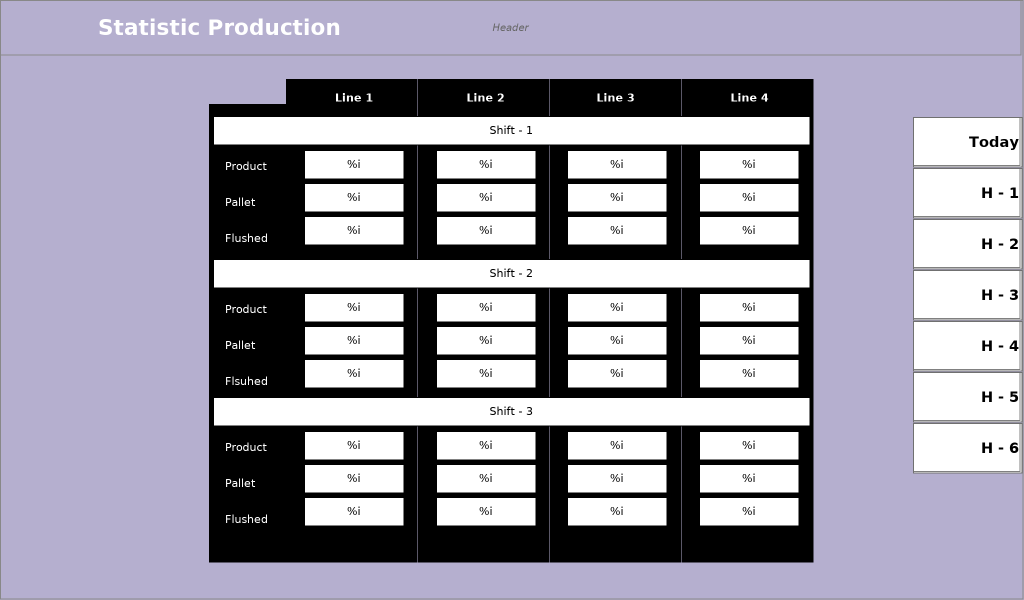
VISUALIZATION OEE_Counter  // 1024x600
    Frame (0,0 1021x55)
        shows Header()
    Button (913,117 109x50), "Today", image: VisuSymbols.Symbols.CalenderDay
        OnMouseClick: execute {
            Data_GVL.dt_OEECounter[1].HMI_NumberPrev := 0;
            Data_GVL.dt_OEECounter[2].HMI_NumberPrev := 0;
            Data_GVL.dt_OEECounter[3].HMI_NumberPrev := 0;
            Data_GVL.dt_OEECounter[4].HMI_NumberPrev := 0;
        }
    Button (913,168 109x50), "H - 1", image: VisuSymbols.Symbols.CalenderDay
        OnMouseClick: execute {
            Data_GVL.dt_OEECounter[1].HMI_NumberPrev := 1;
            Data_GVL.dt_OEECounter[2].HMI_NumberPrev := 1;
            Data_GVL.dt_OEECounter[3].HMI_NumberPrev := 1;
            Data_GVL.dt_OEECounter[4].HMI_NumberPrev := 1;
        }
    Button (913,219 109x50), "H - 2", image: VisuSymbols.Symbols.CalenderDay
        OnMouseClick: execute {
            Data_GVL.dt_OEECounter[1].HMI_NumberPrev := 2;
            Data_GVL.dt_OEECounter[2].HMI_NumberPrev := 2;
            Data_GVL.dt_OEECounter[3].HMI_NumberPrev := 2;
            Data_GVL.dt_OEECounter[4].HMI_NumberPrev := 2;
        }
    Button (913,270 109x50), "H - 3", image: VisuSymbols.Symbols.CalenderDay
        OnMouseClick: execute {
            Data_GVL.dt_OEECounter[1].HMI_NumberPrev := 3;
            Data_GVL.dt_OEECounter[2].HMI_NumberPrev := 3;
            Data_GVL.dt_OEECounter[3].HMI_NumberPrev := 3;
            Data_GVL.dt_OEECounter[4].HMI_NumberPrev := 3;
        }
    Button (913,321 109x50), "H - 4", image: VisuSymbols.Symbols.CalenderDay
        OnMouseClick: execute {
            Data_GVL.dt_OEECounter[1].HMI_NumberPrev := 4;
            Data_GVL.dt_OEECounter[2].HMI_NumberPrev := 4;
            Data_GVL.dt_OEECounter[3].HMI_NumberPrev := 4;
            Data_GVL.dt_OEECounter[4].HMI_NumberPrev := 4;
        }
    Button (913,372 109x50), "H - 5", image: VisuSymbols.Symbols.CalenderDay
        OnMouseClick: execute {
            Data_GVL.dt_OEECounter[1].HMI_NumberPrev := 5;
            Data_GVL.dt_OEECounter[2].HMI_NumberPrev := 5;
            Data_GVL.dt_OEECounter[3].HMI_NumberPrev := 5;
            Data_GVL.dt_OEECounter[4].HMI_NumberPrev := 5;
        }
    Button (913,423 109x50), "H - 6", image: VisuSymbols.Symbols.CalenderDay
        OnMouseClick: execute {
            Data_GVL.dt_OEECounter[1].HMI_NumberPrev := 6;
            Data_GVL.dt_OEECounter[2].HMI_NumberPrev := 6;
            Data_GVL.dt_OEECounter[3].HMI_NumberPrev := 6;
            Data_GVL.dt_OEECounter[4].HMI_NumberPrev := 6;
        }
    Label (95,15 240x25), "Statistic Production"
    RoundedRectangle (286,79 131x483)
    RoundedRectangle (418,79 131x483)
    RoundedRectangle (682,79 131x483)
    RoundedRectangle (550,79 131x483)
    RoundedRectangle (209,104 207x458)
    RoundedRectangle (213,116 597x29), "Shift - 1"
    Label (312,78 84x40), "Line 1"
    Label (222,149 78x35), "Product"
    Label (222,185 78x35), "Pallet"
    Label (222,221 78x35), "Flushed"
    RoundedRectangle (304,150 100x29), "%i", text variable: Data_GVL.dt_OEECounter[1].HMI_Counter[0].Data1
    RoundedRectangle (304,183 100x29), "%i", text variable: Data_GVL.dt_OEECounter[1].HMI_Counter[0].Data2
    RoundedRectangle (304,216 100x29), "%i", text variable: Data_GVL.dt_OEECounter[1].HMI_Counter[0].Data3
    RoundedRectangle (213,259 597x29), "Shift - 2"
    Label (222,292 78x35), "Product"
    Label (222,328 78x35), "Pallet"
    Label (222,364 78x35), "Flsuhed"
    RoundedRectangle (304,293 100x29), "%i", text variable: Data_GVL.dt_OEECounter[1].HMI_Counter[1].Data1
    RoundedRectangle (304,326 100x29), "%i", text variable: Data_GVL.dt_OEECounter[1].HMI_Counter[1].Data2
    RoundedRectangle (304,359 100x29), "%i", text variable: Data_GVL.dt_OEECounter[1].HMI_Counter[1].Data3
    RoundedRectangle (213,397 597x29), "Shift - 3"
    Label (222,430 78x35), "Product"
    Label (222,466 78x35), "Pallet"
    Label (222,502 78x35), "Flushed"
    RoundedRectangle (304,431 100x29), "%i", text variable: Data_GVL.dt_OEECounter[1].HMI_Counter[2].Data1
    RoundedRectangle (304,464 100x29), "%i", text variable: Data_GVL.dt_OEECounter[1].HMI_Counter[2].Data2
    RoundedRectangle (304,497 100x29), "%i", text variable: Data_GVL.dt_OEECounter[1].HMI_Counter[2].Data3
    Label (438,78 95x40), "Line 2"
    RoundedRectangle (436,150 100x29), "%i", text variable: Data_GVL.dt_OEECounter[2].HMI_Counter[0].Data1
    RoundedRectangle (436,183 100x29), "%i", text variable: Data_GVL.dt_OEECounter[2].HMI_Counter[0].Data2
    RoundedRectangle (436,216 100x29), "%i", text variable: Data_GVL.dt_OEECounter[2].HMI_Counter[0].Data3
    RoundedRectangle (436,293 100x29), "%i", text variable: Data_GVL.dt_OEECounter[2].HMI_Counter[1].Data1
    RoundedRectangle (436,326 100x29), "%i", text variable: Data_GVL.dt_OEECounter[2].HMI_Counter[1].Data2
    RoundedRectangle (436,359 100x29), "%i", text variable: Data_GVL.dt_OEECounter[2].HMI_Counter[1].Data3
    RoundedRectangle (436,431 100x29), "%i", text variable: Data_GVL.dt_OEECounter[2].HMI_Counter[2].Data1
    RoundedRectangle (436,464 100x29), "%i", text variable: Data_GVL.dt_OEECounter[2].HMI_Counter[2].Data2
    RoundedRectangle (436,497 100x29), "%i", text variable: Data_GVL.dt_OEECounter[2].HMI_Counter[2].Data3
    RoundedRectangle (567,150 100x29), "%i", text variable: Data_GVL.dt_OEECounter[3].HMI_Counter[0].Data1
    RoundedRectangle (567,183 100x29), "%i", text variable: Data_GVL.dt_OEECounter[3].HMI_Counter[0].Data2
    RoundedRectangle (567,216 100x29), "%i", text variable: Data_GVL.dt_OEECounter[3].HMI_Counter[0].Data3
    RoundedRectangle (567,293 100x29), "%i", text variable: Data_GVL.dt_OEECounter[3].HMI_Counter[1].Data1
    RoundedRectangle (567,326 100x29), "%i", text variable: Data_GVL.dt_OEECounter[3].HMI_Counter[1].Data2
    RoundedRectangle (567,359 100x29), "%i", text variable: Data_GVL.dt_OEECounter[3].HMI_Counter[1].Data3
    RoundedRectangle (567,431 100x29), "%i", text variable: Data_GVL.dt_OEECounter[3].HMI_Counter[2].Data1
    RoundedRectangle (567,464 100x29), "%i", text variable: Data_GVL.dt_OEECounter[3].HMI_Counter[2].Data2
    RoundedRectangle (567,497 100x29), "%i", text variable: Data_GVL.dt_OEECounter[3].HMI_Counter[2].Data3
    RoundedRectangle (699,150 100x29), "%i", text variable: Data_GVL.dt_OEECounter[4].HMI_Counter[0].Data1
    RoundedRectangle (699,183 100x29), "%i", text variable: Data_GVL.dt_OEECounter[4].HMI_Counter[0].Data2
    RoundedRectangle (699,216 100x29), "%i", text variable: Data_GVL.dt_OEECounter[4].HMI_Counter[0].Data3
    RoundedRectangle (699,293 100x29), "%i", text variable: Data_GVL.dt_OEECounter[4].HMI_Counter[1].Data1
    RoundedRectangle (699,326 100x29), "%i", text variable: Data_GVL.dt_OEECounter[4].HMI_Counter[1].Data2
    RoundedRectangle (699,359 100x29), "%i", text variable: Data_GVL.dt_OEECounter[4].HMI_Counter[1].Data3
    RoundedRectangle (699,431 100x29), "%i", text variable: Data_GVL.dt_OEECounter[4].HMI_Counter[2].Data1
    RoundedRectangle (699,464 100x29), "%i", text variable: Data_GVL.dt_OEECounter[4].HMI_Counter[2].Data2
    RoundedRectangle (699,497 100x29), "%i", text variable: Data_GVL.dt_OEECounter[4].HMI_Counter[2].Data3
    Label (568,78 95x40), "Line 3"
    Label (702,78 95x40), "Line 4"
END_VISUALIZATION

(* stored: Version 1.1.0.1, ProductVersion 3.1.4024.12
   Visu OEE_Counter: Id {3aa3e7b6-5ff8-446f-8f20-b94430ea3f6b} *)
